PROGRAM Motor_Example
VAR
	TON_TEST: TON;
	TON_TEST_PT: TIME := T#60S;
	TON_TEST_ET: TIME;
	TON_TEST_TRIGGER : BOOL;
	TON_TEST_ET_SAV: TIME;
	Not_Equal_Zero : TIME :=T#0s;
END_VAR

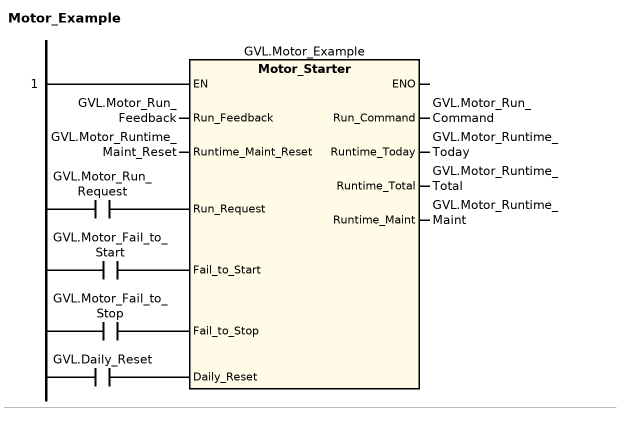
// NETWORK 1
GVL.Motor_Example(
    Run_Feedback := GVL.Motor_Run_Feedback,
    Runtime_Maint_Reset := GVL.Motor_Runtime_Maint_Reset,
    Run_Request := GVL.Motor_Run_Request,
    Fail_to_Start := GVL.Motor_Fail_to_Start,
    Fail_to_Stop := GVL.Motor_Fail_to_Stop,
    Daily_Reset := GVL.Daily_Reset,
    Run_Command => GVL.Motor_Run_Command,
    Runtime_Today => GVL.Motor_Runtime_Today,
    Runtime_Total => GVL.Motor_Runtime_Total,
    Runtime_Maint => GVL.Motor_Runtime_Maint); // Motor_Starter

END_PROGRAM

(* stored: Version 1.1.0.1, ProductVersion 3.1.4024.12
   POU Motor_Example: Id {875228a8-8d81-4320-b913-8585bf7e4dcc}, SpecialFunc None *)
